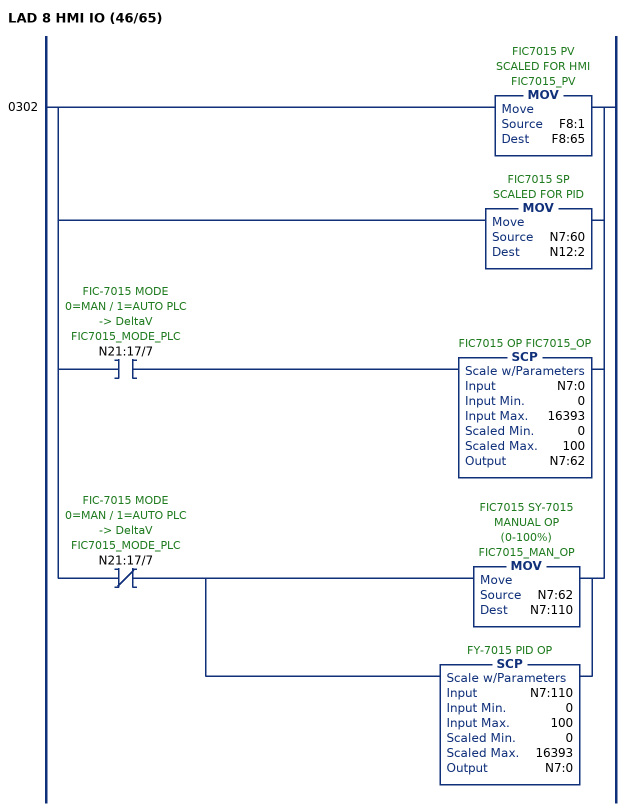
% Rung: 302 %
SOR BST MOV F8:1 F8:65 NXB MOV N7:60 N12:2 NXB XIC N21:17/7 SCP N7:0 0 16393 0 100 N7:62 NXB XIO N21:17/7 BST MOV N7:62 N7:110 NXB SCP N7:110 0 100 0 16393 N7:0 BND BND EOR
%   F8:1  FT_7010_SCI  "FT-7010 SCALED INPUT" %
%   F8:65  FIC7015_PV  "FIC7015 PV SCALED FOR HMI" %
%   N7:60  FIC7015_SP  "FIC7015 SP" %
%   N12:2  "FIC7015 SP SCALED FOR PID" %
%   N21:17/7  FIC7015_MODE_PLC  "FIC-7015 MODE 0=MAN / 1=AUTO PLC -> DeltaV" %
%   N7:0  "FY-7015 PID OP" %
%   N7:62  FIC7015_OP  "FIC7015 OP" %
%   N7:110  FIC7015_MAN_OP  "FIC7015 SY-7015 MANUAL OP (0-100%)" %

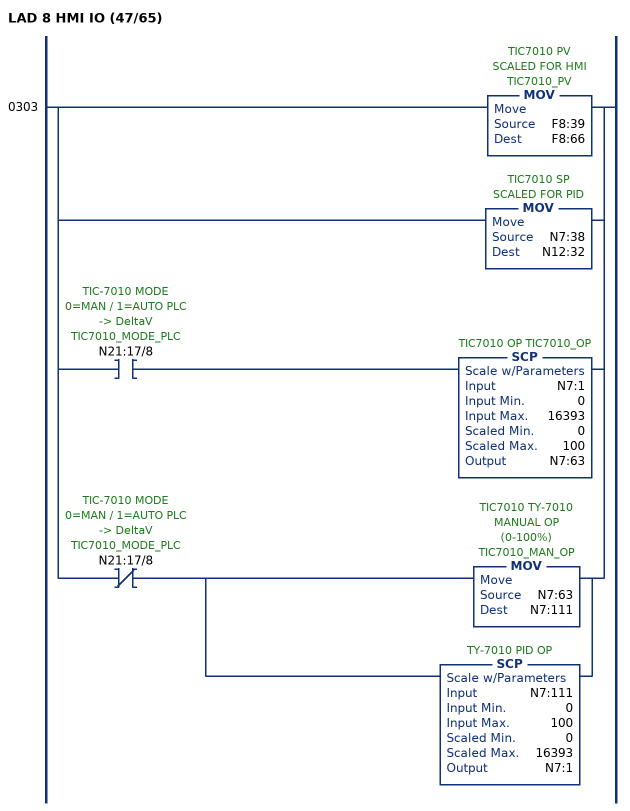
% Rung: 303 %
SOR BST MOV F8:39 F8:66 NXB MOV N7:38 N12:32 NXB XIC N21:17/8 SCP N7:1 0 16393 0 100 N7:63 NXB XIO N21:17/8 BST MOV N7:63 N7:111 NXB SCP N7:111 0 100 0 16393 N7:1 BND BND EOR
%   F8:39  TT_7010_SCI  "TT-7010 SCALED INPUT" %
%   F8:66  TIC7010_PV  "TIC7010 PV SCALED FOR HMI" %
%   N7:38  TIC7010_SP  "TIC7010 SP" %
%   N12:32  "TIC7010 SP SCALED FOR PID" %
%   N21:17/8  TIC7010_MODE_PLC  "TIC-7010 MODE 0=MAN / 1=AUTO PLC -> DeltaV" %
%   N7:1  "TY-7010 PID OP" %
%   N7:63  TIC7010_OP  "TIC7010 OP" %
%   N7:111  TIC7010_MAN_OP  "TIC7010 TY-7010 MANUAL OP (0-100%)" %

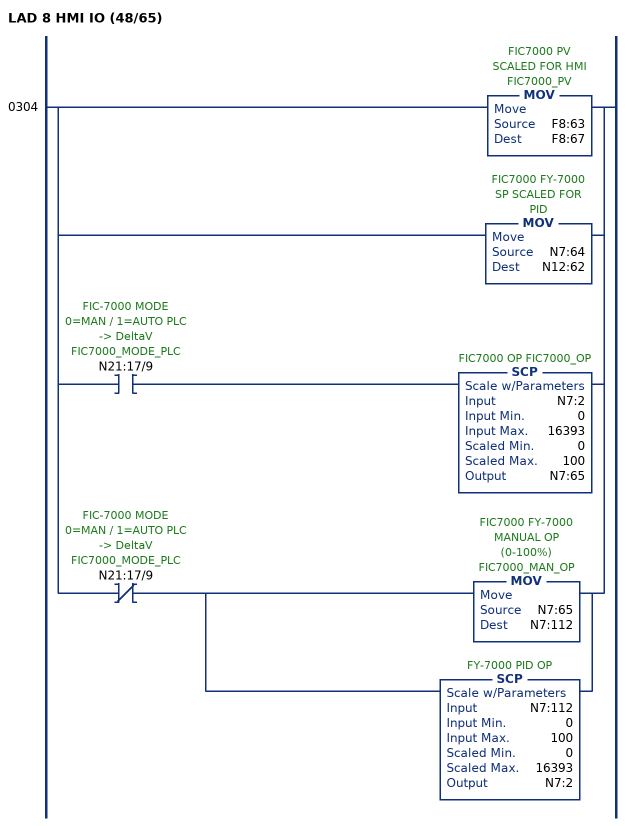
% Rung: 304 %
SOR BST MOV F8:63 F8:67 NXB MOV N7:64 N12:62 NXB XIC N21:17/9 SCP N7:2 0 16393 0 100 N7:65 NXB XIO N21:17/9 BST MOV N7:65 N7:112 NXB SCP N7:112 0 100 0 16393 N7:2 BND BND EOR
%   F8:63  PT_7026_SCI  "PT-7026 SCALED INPUT" %
%   F8:67  FIC7000_PV  "FIC7000 PV SCALED FOR HMI" %
%   N7:64  FIC7000_SP  "FIC7000 SP" %
%   N12:62  "FIC7000 FY-7000 SP SCALED FOR PID" %
%   N21:17/9  FIC7000_MODE_PLC  "FIC-7000 MODE 0=MAN / 1=AUTO PLC -> DeltaV" %
%   N7:2  "FY-7000 PID OP" %
%   N7:65  FIC7000_OP  "FIC7000 OP" %
%   N7:112  FIC7000_MAN_OP  "FIC7000 FY-7000 MANUAL OP (0-100%)" %

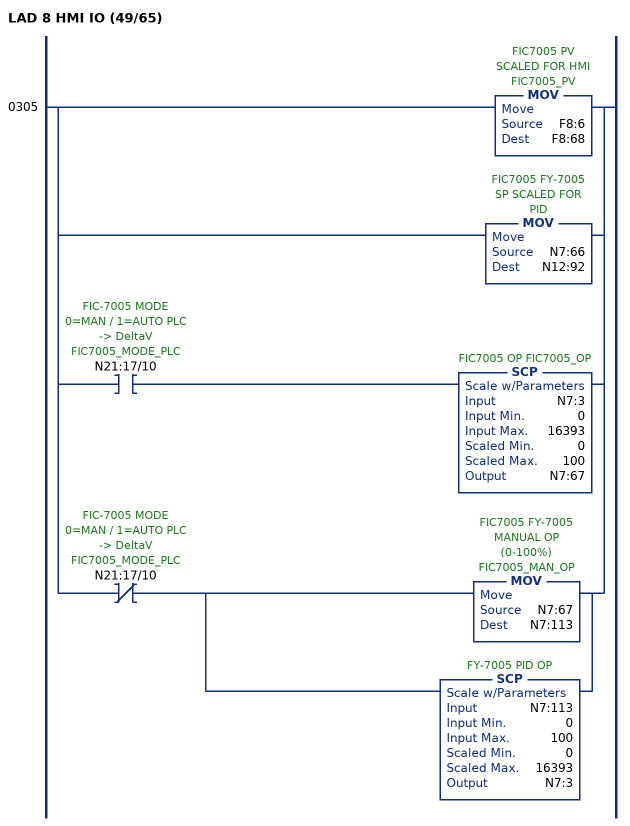
% Rung: 305 %
SOR BST MOV F8:6 F8:68 NXB MOV N7:66 N12:92 NXB XIC N21:17/10 SCP N7:3 0 16393 0 100 N7:67 NXB XIO N21:17/10 BST MOV N7:67 N7:113 NXB SCP N7:113 0 100 0 16393 N7:3 BND BND EOR
%   F8:6  FT_7005_SCI  "FT-7005 SCALED INPUT" %
%   F8:68  FIC7005_PV  "FIC7005 PV SCALED FOR HMI" %
%   N7:66  FIC7005_SP  "FIC7005 SP" %
%   N12:92  "FIC7005 FY-7005 SP SCALED FOR PID" %
%   N21:17/10  FIC7005_MODE_PLC  "FIC-7005 MODE 0=MAN / 1=AUTO PLC -> DeltaV" %
%   N7:3  "FY-7005 PID OP" %
%   N7:67  FIC7005_OP  "FIC7005 OP" %
%   N7:113  FIC7005_MAN_OP  "FIC7005 FY-7005 MANUAL OP (0-100%)" %

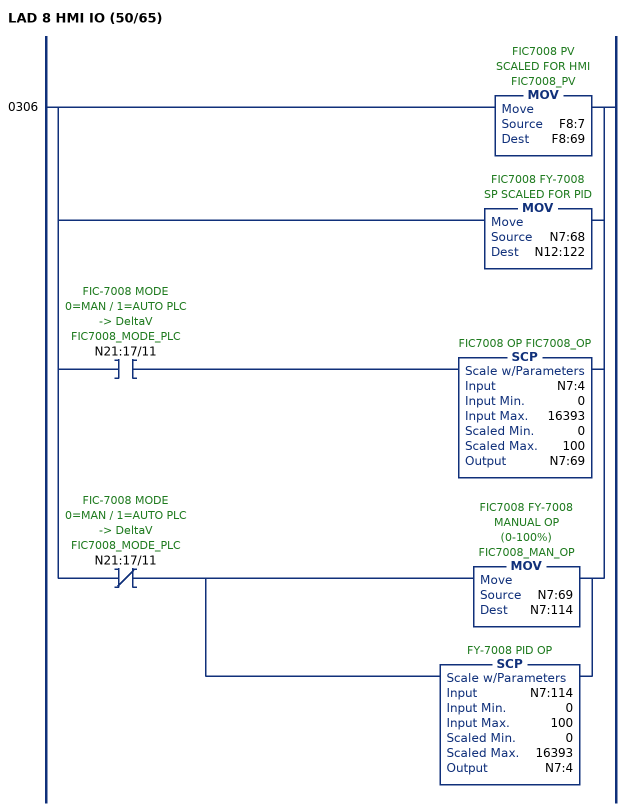
% Rung: 306 %
SOR BST MOV F8:7 F8:69 NXB MOV N7:68 N12:122 NXB XIC N21:17/11 SCP N7:4 0 16393 0 100 N7:69 NXB XIO N21:17/11 BST MOV N7:69 N7:114 NXB SCP N7:114 0 100 0 16393 N7:4 BND BND EOR
%   F8:7  FT_7008_SCI  "FT-7008 SCALED INPUT" %
%   F8:69  FIC7008_PV  "FIC7008 PV SCALED FOR HMI" %
%   N7:68  FIC7008_SP  "FIC7008 SP" %
%   N12:122  "FIC7008 FY-7008 SP SCALED FOR PID" %
%   N21:17/11  FIC7008_MODE_PLC  "FIC-7008 MODE 0=MAN / 1=AUTO PLC -> DeltaV" %
%   N7:4  "FY-7008 PID OP" %
%   N7:69  FIC7008_OP  "FIC7008 OP" %
%   N7:114  FIC7008_MAN_OP  "FIC7008 FY-7008 MANUAL OP (0-100%)" %

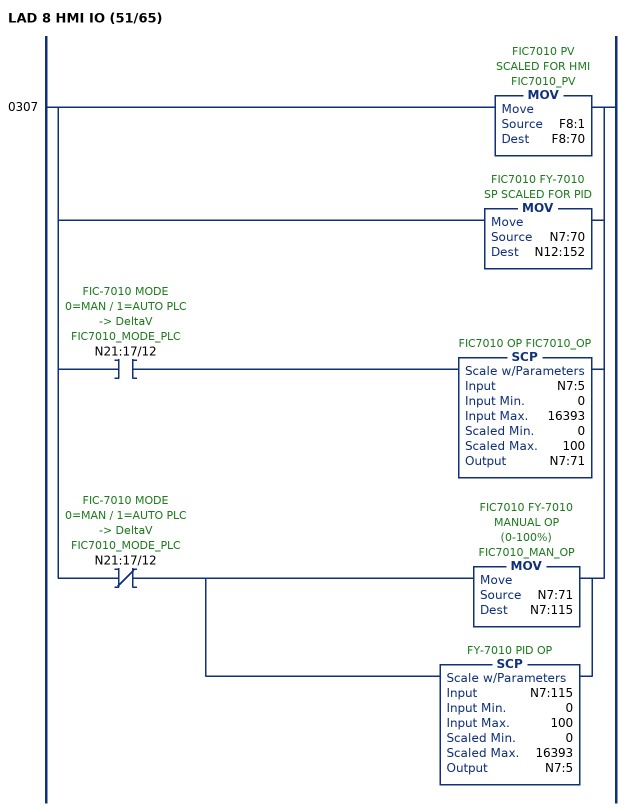
% Rung: 307 %
SOR BST MOV F8:1 F8:70 NXB MOV N7:70 N12:152 NXB XIC N21:17/12 SCP N7:5 0 16393 0 100 N7:71 NXB XIO N21:17/12 BST MOV N7:71 N7:115 NXB SCP N7:115 0 100 0 16393 N7:5 BND BND EOR
%   F8:1  FT_7010_SCI  "FT-7010 SCALED INPUT" %
%   F8:70  FIC7010_PV  "FIC7010 PV SCALED FOR HMI" %
%   N7:70  FIC7010_SP  "FIC7010 SP" %
%   N12:152  "FIC7010 FY-7010 SP SCALED FOR PID" %
%   N21:17/12  FIC7010_MODE_PLC  "FIC-7010 MODE 0=MAN / 1=AUTO PLC -> DeltaV" %
%   N7:5  "FY-7010 PID OP" %
%   N7:71  FIC7010_OP  "FIC7010 OP" %
%   N7:115  FIC7010_MAN_OP  "FIC7010 FY-7010 MANUAL OP (0-100%)" %

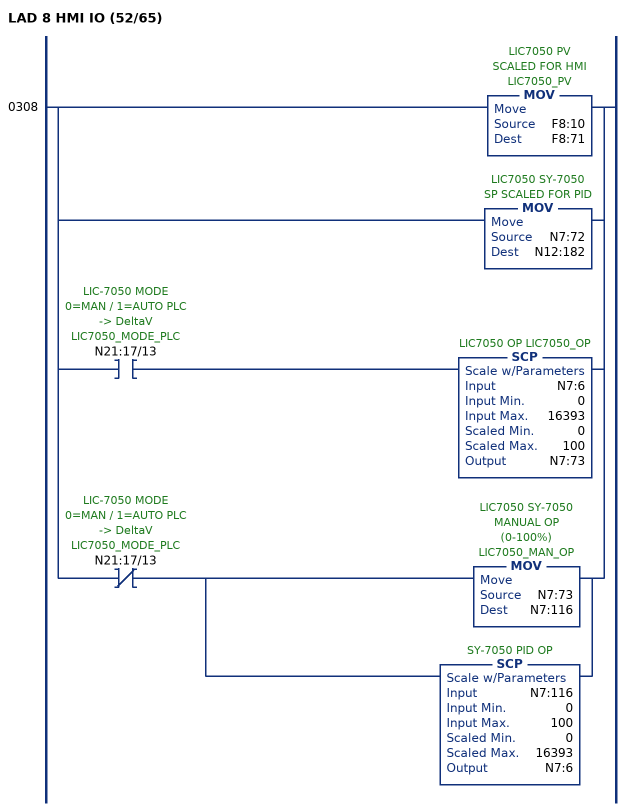
% Rung: 308 %
SOR BST MOV F8:10 F8:71 NXB MOV N7:72 N12:182 NXB XIC N21:17/13 SCP N7:6 0 16393 0 100 N7:73 NXB XIO N21:17/13 BST MOV N7:73 N7:116 NXB SCP N7:116 0 100 0 16393 N7:6 BND BND EOR
%   F8:10  LT_7050_SCI  "LT-7050 SCALED INPUT" %
%   F8:71  LIC7050_PV  "LIC7050 PV SCALED FOR HMI" %
%   N7:72  LIC7050_SP  "LIC7050 SP" %
%   N12:182  "LIC7050 SY-7050 SP SCALED FOR PID" %
%   N21:17/13  LIC7050_MODE_PLC  "LIC-7050 MODE 0=MAN / 1=AUTO PLC -> DeltaV" %
%   N7:6  "SY-7050 PID OP" %
%   N7:73  LIC7050_OP  "LIC7050 OP" %
%   N7:116  LIC7050_MAN_OP  "LIC7050 SY-7050 MANUAL OP (0-100%)" %

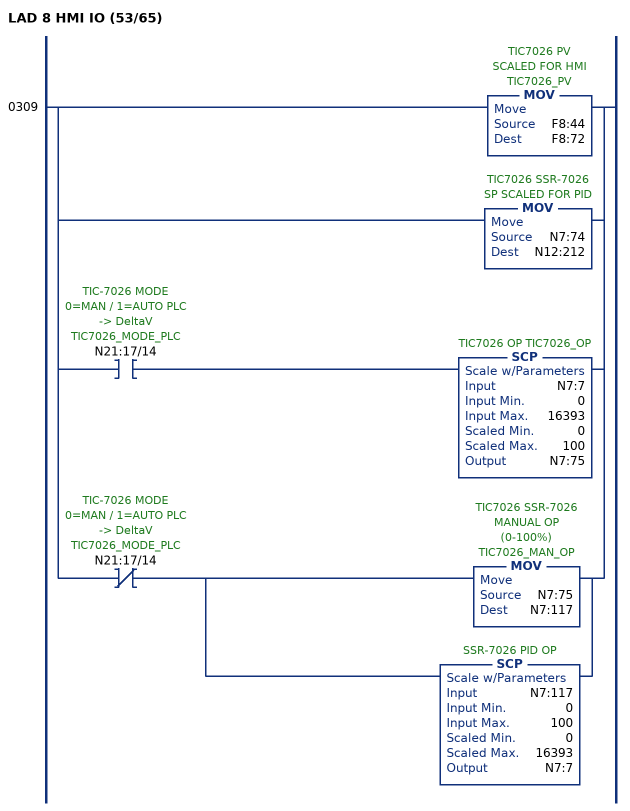
% Rung: 309 %
SOR BST MOV F8:44 F8:72 NXB MOV N7:74 N12:212 NXB XIC N21:17/14 SCP N7:7 0 16393 0 100 N7:75 NXB XIO N21:17/14 BST MOV N7:75 N7:117 NXB SCP N7:117 0 100 0 16393 N7:7 BND BND EOR
%   F8:44  TT_7026_SCI  "TT-7026 SCALED INPUT" %
%   F8:72  TIC7026_PV  "TIC7026 PV SCALED FOR HMI" %
%   N7:74  TIC7026_SP  "TIC7026 SP" %
%   N12:212  "TIC7026 SSR-7026 SP SCALED FOR PID" %
%   N21:17/14  TIC7026_MODE_PLC  "TIC-7026 MODE 0=MAN / 1=AUTO PLC -> DeltaV" %
%   N7:7  "SSR-7026 PID OP" %
%   N7:75  TIC7026_OP  "TIC7026 OP" %
%   N7:117  TIC7026_MAN_OP  "TIC7026 SSR-7026 MANUAL OP (0-100%)" %

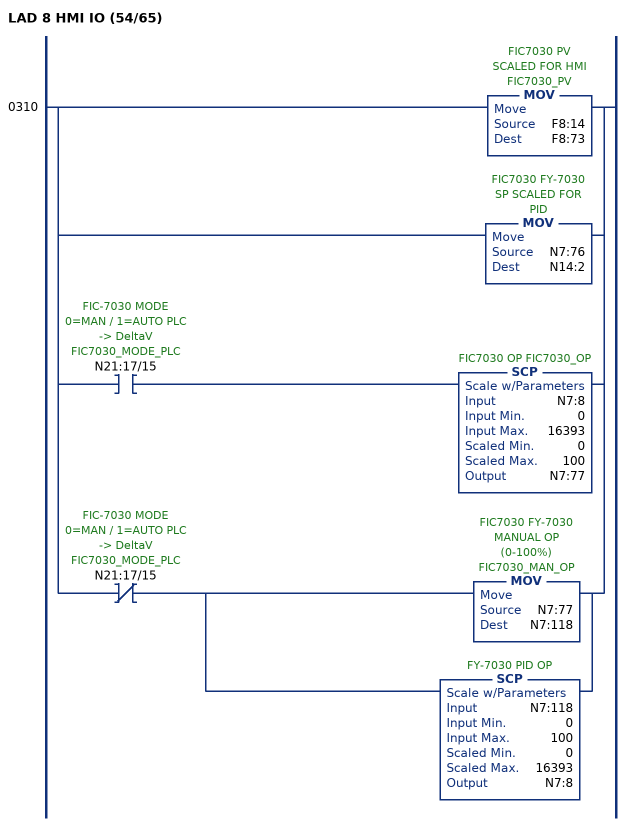
% Rung: 310 %
SOR BST MOV F8:14 F8:73 NXB MOV N7:76 N14:2 NXB XIC N21:17/15 SCP N7:8 0 16393 0 100 N7:77 NXB XIO N21:17/15 BST MOV N7:77 N7:118 NXB SCP N7:118 0 100 0 16393 N7:8 BND BND EOR
%   F8:14  FT_7030_SCI  "FT-7030 SCALED INPUT" %
%   F8:73  FIC7030_PV  "FIC7030 PV SCALED FOR HMI" %
%   N7:76  FIC7030_SP  "FIC7030 SP" %
%   N14:2  "FIC7030 FY-7030 SP SCALED FOR PID" %
%   N21:17/15  FIC7030_MODE_PLC  "FIC-7030 MODE 0=MAN / 1=AUTO PLC -> DeltaV" %
%   N7:8  "FY-7030 PID OP" %
%   N7:77  FIC7030_OP  "FIC7030 OP" %
%   N7:118  FIC7030_MAN_OP  "FIC7030 FY-7030 MANUAL OP (0-100%)" %

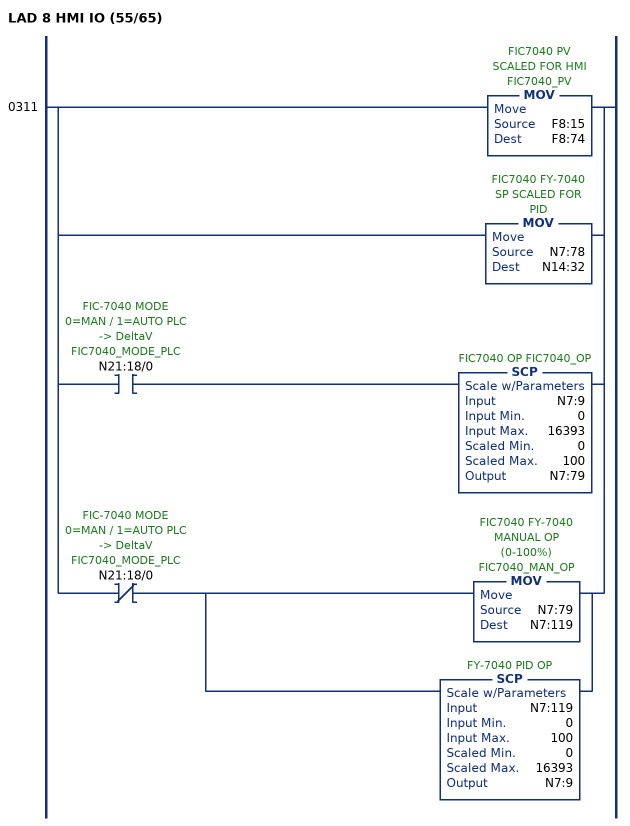
% Rung: 311 %
SOR BST MOV F8:15 F8:74 NXB MOV N7:78 N14:32 NXB XIC N21:18/0 SCP N7:9 0 16393 0 100 N7:79 NXB XIO N21:18/0 BST MOV N7:79 N7:119 NXB SCP N7:119 0 100 0 16393 N7:9 BND BND EOR
%   F8:15  FT_7040_SCI  "FT-7040 SCALED INPUT" %
%   F8:74  FIC7040_PV  "FIC7040 PV SCALED FOR HMI" %
%   N7:78  FIC7040_SP  "FIC7040 SP" %
%   N14:32  "FIC7040 FY-7040 SP SCALED FOR PID" %
%   N21:18/0  FIC7040_MODE_PLC  "FIC-7040 MODE 0=MAN / 1=AUTO PLC -> DeltaV" %
%   N7:9  "FY-7040 PID OP" %
%   N7:79  FIC7040_OP  "FIC7040 OP" %
%   N7:119  FIC7040_MAN_OP  "FIC7040 FY-7040 MANUAL OP (0-100%)" %

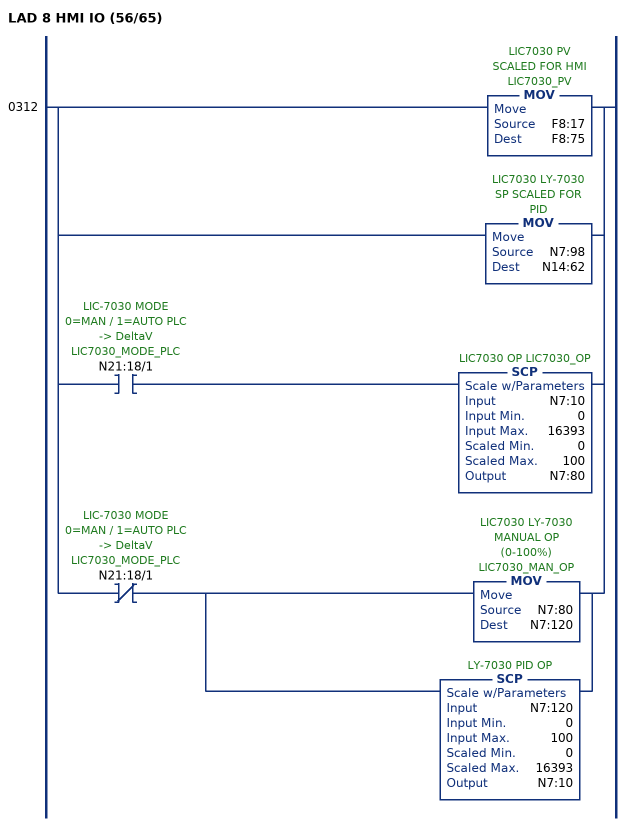
% Rung: 312 %
SOR BST MOV F8:17 F8:75 NXB MOV N7:98 N14:62 NXB XIC N21:18/1 SCP N7:10 0 16393 0 100 N7:80 NXB XIO N21:18/1 BST MOV N7:80 N7:120 NXB SCP N7:120 0 100 0 16393 N7:10 BND BND EOR
%   F8:17  LT_7030_SCI  "LT-7030 SCALED INPUT" %
%   F8:75  LIC7030_PV  "LIC7030 PV SCALED FOR HMI" %
%   N7:98  LIC7030_SP  "LIC7030 SP" %
%   N14:62  "LIC7030 LY-7030 SP SCALED FOR PID" %
%   N21:18/1  LIC7030_MODE_PLC  "LIC-7030 MODE 0=MAN / 1=AUTO PLC -> DeltaV" %
%   N7:10  "LY-7030 PID OP" %
%   N7:80  LIC7030_OP  "LIC7030 OP" %
%   N7:120  LIC7030_MAN_OP  "LIC7030 LY-7030 MANUAL OP (0-100%)" %

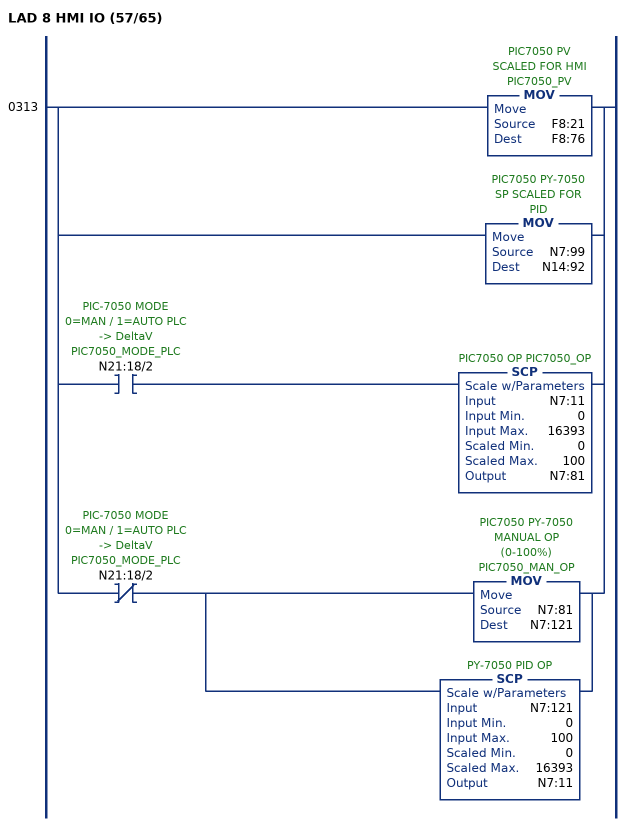
% Rung: 313 %
SOR BST MOV F8:21 F8:76 NXB MOV N7:99 N14:92 NXB XIC N21:18/2 SCP N7:11 0 16393 0 100 N7:81 NXB XIO N21:18/2 BST MOV N7:81 N7:121 NXB SCP N7:121 0 100 0 16393 N7:11 BND BND EOR
%   F8:21  PT_7050_SCI  "PT-7050 SCALED INPUT" %
%   F8:76  PIC7050_PV  "PIC7050 PV SCALED FOR HMI" %
%   N7:99  PIC7050_SP  "PIC7050 SP" %
%   N14:92  "PIC7050 PY-7050 SP SCALED FOR PID" %
%   N21:18/2  PIC7050_MODE_PLC  "PIC-7050 MODE 0=MAN / 1=AUTO PLC -> DeltaV" %
%   N7:11  "PY-7050 PID OP" %
%   N7:81  PIC7050_OP  "PIC7050 OP" %
%   N7:121  PIC7050_MAN_OP  "PIC7050 PY-7050 MANUAL OP (0-100%)" %

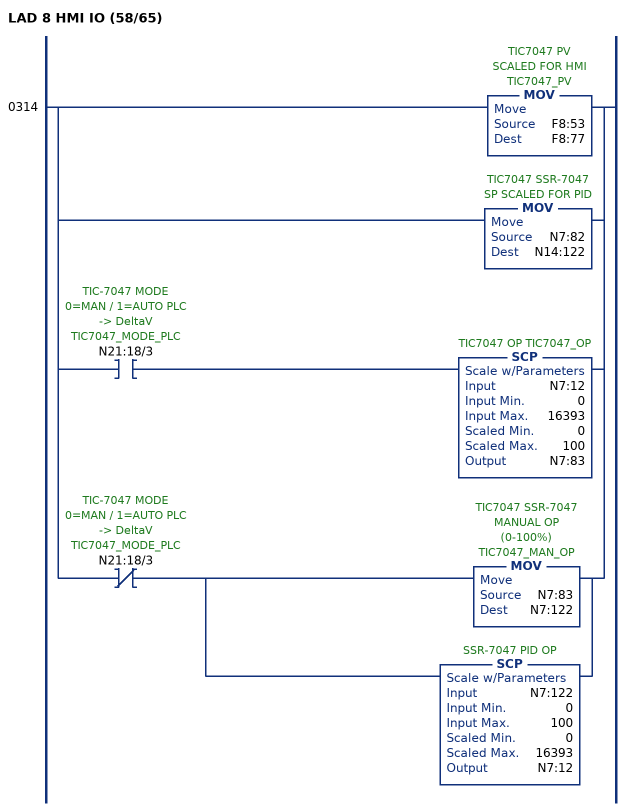
% Rung: 314 %
SOR BST MOV F8:53 F8:77 NXB MOV N7:82 N14:122 NXB XIC N21:18/3 SCP N7:12 0 16393 0 100 N7:83 NXB XIO N21:18/3 BST MOV N7:83 N7:122 NXB SCP N7:122 0 100 0 16393 N7:12 BND BND EOR
%   F8:53  TT_7047_SCI  "TT-7047 SCALED INPUT" %
%   F8:77  TIC7047_PV  "TIC7047 PV SCALED FOR HMI" %
%   N7:82  TIC7047_SP  "TIC7047 SP" %
%   N14:122  "TIC7047 SSR-7047 SP SCALED FOR PID" %
%   N21:18/3  TIC7047_MODE_PLC  "TIC-7047 MODE 0=MAN / 1=AUTO PLC -> DeltaV" %
%   N7:12  "SSR-7047 PID OP" %
%   N7:83  TIC7047_OP  "TIC7047 OP" %
%   N7:122  TIC7047_MAN_OP  "TIC7047 SSR-7047 MANUAL OP (0-100%)" %

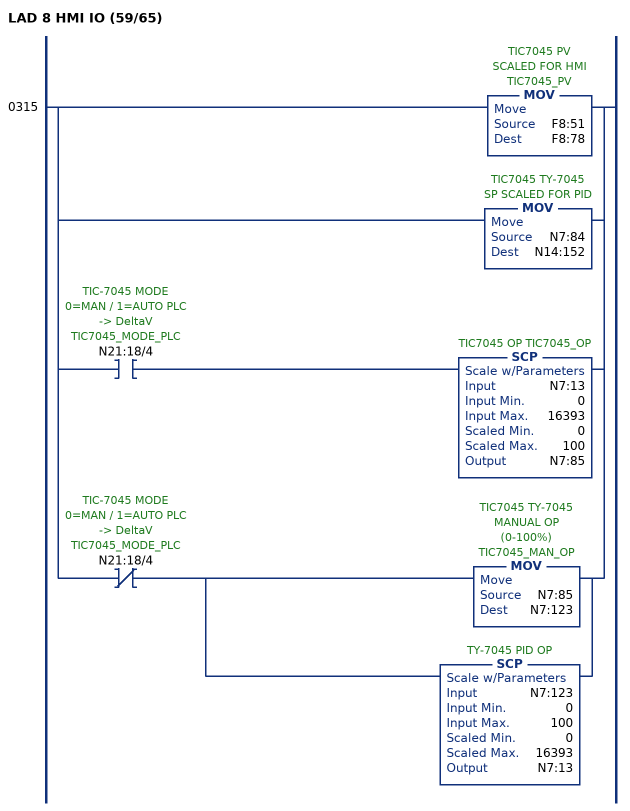
% Rung: 315 %
SOR BST MOV F8:51 F8:78 NXB MOV N7:84 N14:152 NXB XIC N21:18/4 SCP N7:13 0 16393 0 100 N7:85 NXB XIO N21:18/4 BST MOV N7:85 N7:123 NXB SCP N7:123 0 100 0 16393 N7:13 BND BND EOR
%   F8:51  TT_7045_SCI  "TT-7045 SCALED INPUT" %
%   F8:78  TIC7045_PV  "TIC7045 PV SCALED FOR HMI" %
%   N7:84  TIC7045_SP  "TIC7045 SP" %
%   N14:152  "TIC7045 TY-7045 SP SCALED FOR PID" %
%   N21:18/4  TIC7045_MODE_PLC  "TIC-7045 MODE 0=MAN / 1=AUTO PLC -> DeltaV" %
%   N7:13  "TY-7045 PID OP" %
%   N7:85  TIC7045_OP  "TIC7045 OP" %
%   N7:123  TIC7045_MAN_OP  "TIC7045 TY-7045 MANUAL OP (0-100%)" %

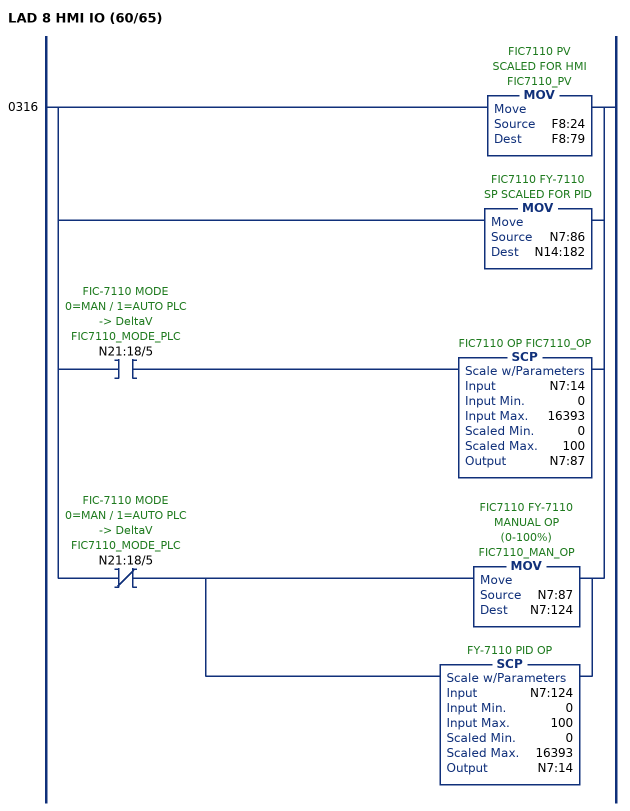
% Rung: 316 %
SOR BST MOV F8:24 F8:79 NXB MOV N7:86 N14:182 NXB XIC N21:18/5 SCP N7:14 0 16393 0 100 N7:87 NXB XIO N21:18/5 BST MOV N7:87 N7:124 NXB SCP N7:124 0 100 0 16393 N7:14 BND BND EOR
%   F8:24  FT_7110_SCI  "FT-7110 SCALED INPUT" %
%   F8:79  FIC7110_PV  "FIC7110 PV SCALED FOR HMI" %
%   N7:86  FIC7110_SP  "FIC7110 SP" %
%   N14:182  "FIC7110 FY-7110 SP SCALED FOR PID" %
%   N21:18/5  FIC7110_MODE_PLC  "FIC-7110 MODE 0=MAN / 1=AUTO PLC -> DeltaV" %
%   N7:14  "FY-7110 PID OP" %
%   N7:87  FIC7110_OP  "FIC7110 OP" %
%   N7:124  FIC7110_MAN_OP  "FIC7110 FY-7110 MANUAL OP (0-100%)" %

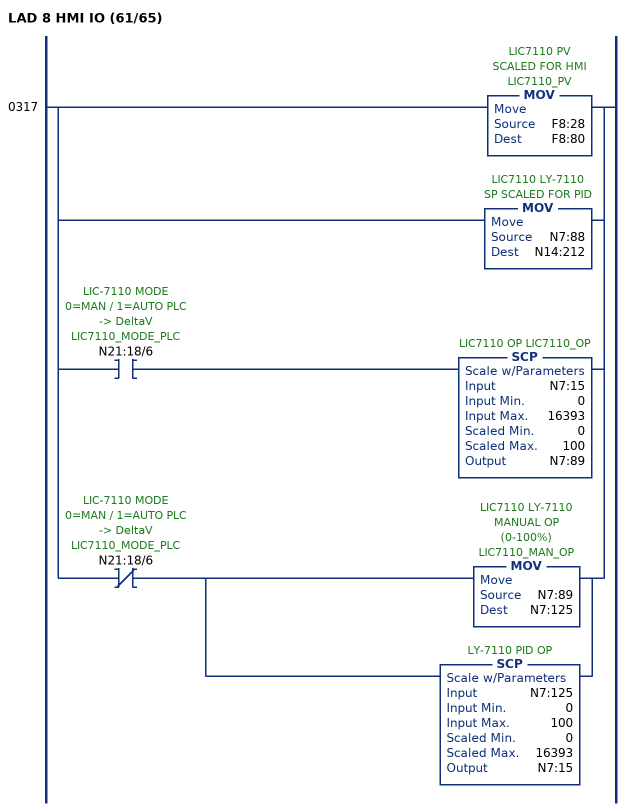
% Rung: 317 %
SOR BST MOV F8:28 F8:80 NXB MOV N7:88 N14:212 NXB XIC N21:18/6 SCP N7:15 0 16393 0 100 N7:89 NXB XIO N21:18/6 BST MOV N7:89 N7:125 NXB SCP N7:125 0 100 0 16393 N7:15 BND BND EOR
%   F8:28  LT_7110_SCI  "LT-7110 SCALED INPUT" %
%   F8:80  LIC7110_PV  "LIC7110 PV SCALED FOR HMI" %
%   N7:88  LIC7110_SP  "LIC7110 SP" %
%   N14:212  "LIC7110 LY-7110 SP SCALED FOR PID" %
%   N21:18/6  LIC7110_MODE_PLC  "LIC-7110 MODE 0=MAN / 1=AUTO PLC -> DeltaV" %
%   N7:15  "LY-7110 PID OP" %
%   N7:89  LIC7110_OP  "LIC7110 OP" %
%   N7:125  LIC7110_MAN_OP  "LIC7110 LY-7110 MANUAL OP (0-100%)" %

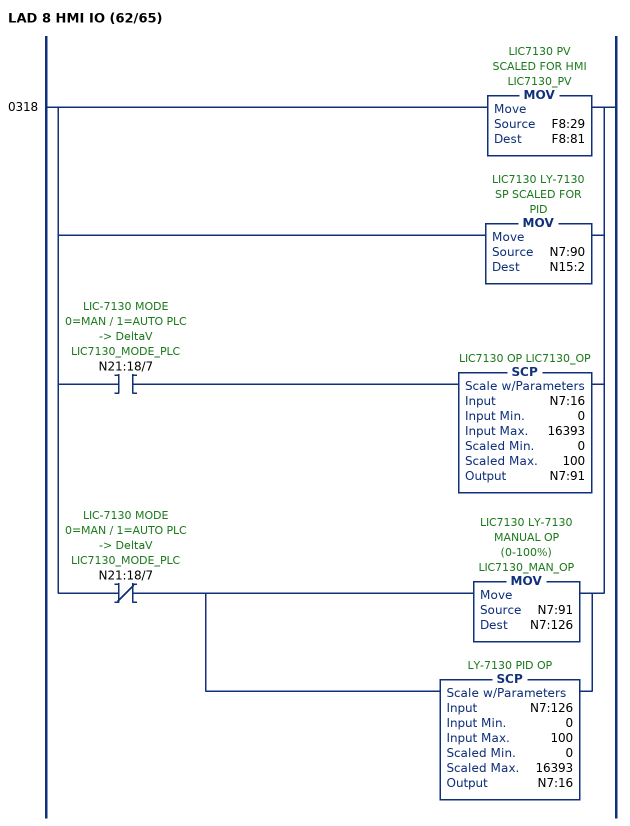
% Rung: 318 %
SOR BST MOV F8:29 F8:81 NXB MOV N7:90 N15:2 NXB XIC N21:18/7 SCP N7:16 0 16393 0 100 N7:91 NXB XIO N21:18/7 BST MOV N7:91 N7:126 NXB SCP N7:126 0 100 0 16393 N7:16 BND BND EOR
%   F8:29  LT_7130_SCI  "LT-7130 SCALED INPUT" %
%   F8:81  LIC7130_PV  "LIC7130 PV SCALED FOR HMI" %
%   N7:90  LIC7130_SP  "LIC7130 SP" %
%   N15:2  "LIC7130 LY-7130 SP SCALED FOR PID" %
%   N21:18/7  LIC7130_MODE_PLC  "LIC-7130 MODE 0=MAN / 1=AUTO PLC -> DeltaV" %
%   N7:16  "LY-7130 PID OP" %
%   N7:91  LIC7130_OP  "LIC7130 OP" %
%   N7:126  LIC7130_MAN_OP  "LIC7130 LY-7130 MANUAL OP (0-100%)" %

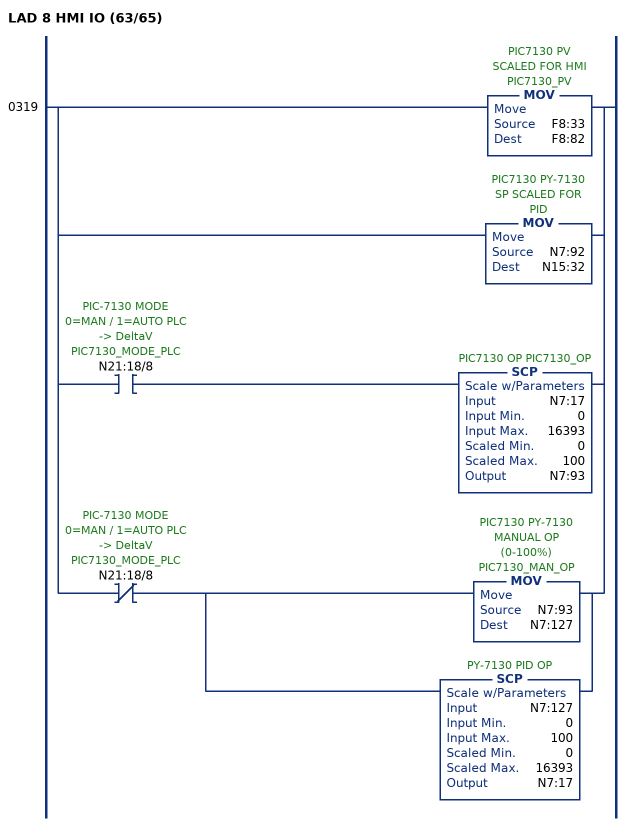
% Rung: 319 %
SOR BST MOV F8:33 F8:82 NXB MOV N7:92 N15:32 NXB XIC N21:18/8 SCP N7:17 0 16393 0 100 N7:93 NXB XIO N21:18/8 BST MOV N7:93 N7:127 NXB SCP N7:127 0 100 0 16393 N7:17 BND BND EOR
%   F8:33  PT_7130_SCI  "PT-7130 SCALED INPUT" %
%   F8:82  PIC7130_PV  "PIC7130 PV SCALED FOR HMI" %
%   N7:92  PIC7130_SP  "PIC7130 SP" %
%   N15:32  "PIC7130 PY-7130 SP SCALED FOR PID" %
%   N21:18/8  PIC7130_MODE_PLC  "PIC-7130 MODE 0=MAN / 1=AUTO PLC -> DeltaV" %
%   N7:17  "PY-7130 PID OP" %
%   N7:93  PIC7130_OP  "PIC7130 OP" %
%   N7:127  PIC7130_MAN_OP  "PIC7130 PY-7130 MANUAL OP (0-100%)" %

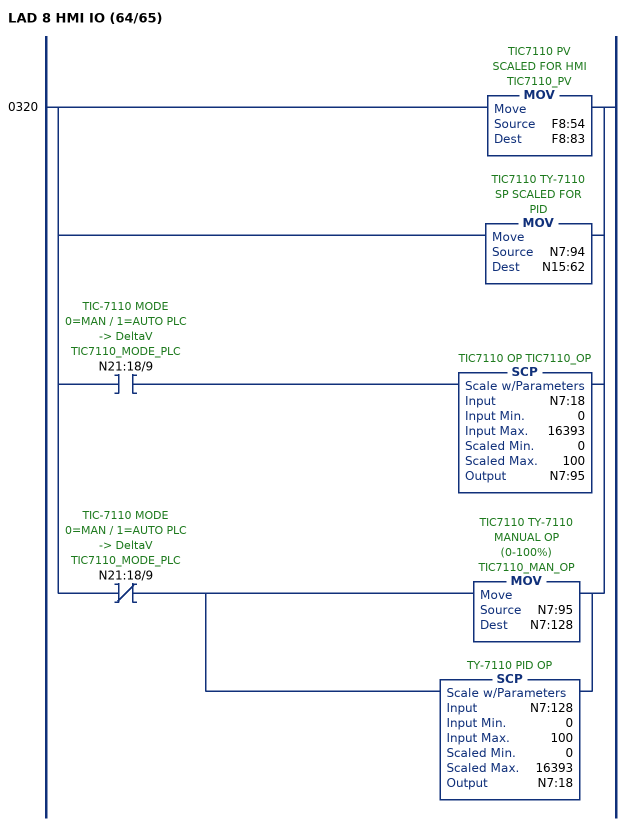
% Rung: 320 %
SOR BST MOV F8:54 F8:83 NXB MOV N7:94 N15:62 NXB XIC N21:18/9 SCP N7:18 0 16393 0 100 N7:95 NXB XIO N21:18/9 BST MOV N7:95 N7:128 NXB SCP N7:128 0 100 0 16393 N7:18 BND BND EOR
%   F8:54  TT_7110_SCI  "TT-7110 SCALED INPUT" %
%   F8:83  TIC7110_PV  "TIC7110 PV SCALED FOR HMI" %
%   N7:94  TIC7110_SP  "TIC7110 SP" %
%   N15:62  "TIC7110 TY-7110 SP SCALED FOR PID" %
%   N21:18/9  TIC7110_MODE_PLC  "TIC-7110 MODE 0=MAN / 1=AUTO PLC -> DeltaV" %
%   N7:18  "TY-7110 PID OP" %
%   N7:95  TIC7110_OP  "TIC7110 OP" %
%   N7:128  TIC7110_MAN_OP  "TIC7110 TY-7110 MANUAL OP (0-100%)" %

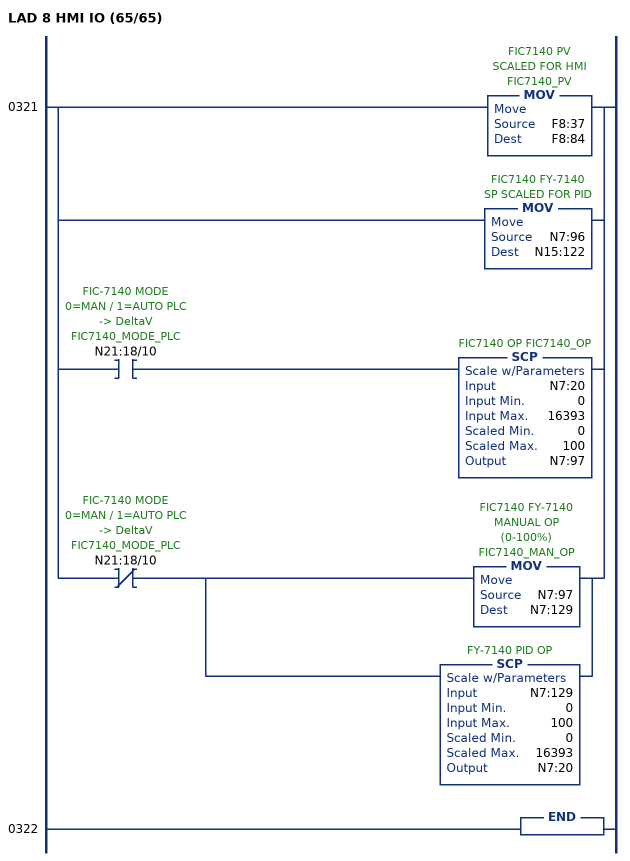
% Rung: 321 %
SOR BST MOV F8:37 F8:84 NXB MOV N7:96 N15:122 NXB XIC N21:18/10 SCP N7:20 0 16393 0 100 N7:97 NXB XIO N21:18/10 BST MOV N7:97 N7:129 NXB SCP N7:129 0 100 0 16393 N7:20 BND BND EOR
%   F8:37  FT_7140_SCI  "FT-7140 SCALED INPUT" %
%   F8:84  FIC7140_PV  "FIC7140 PV SCALED FOR HMI" %
%   N7:96  FIC7140_SP  "FIC7140 SP" %
%   N15:122  "FIC7140 FY-7140 SP SCALED FOR PID" %
%   N21:18/10  FIC7140_MODE_PLC  "FIC-7140 MODE 0=MAN / 1=AUTO PLC -> DeltaV" %
%   N7:20  "FY-7140 PID OP" %
%   N7:97  FIC7140_OP  "FIC7140 OP" %
%   N7:129  FIC7140_MAN_OP  "FIC7140 FY-7140 MANUAL OP (0-100%)" %
% Rung: 322 %
SOR END EOR

LADDER 9 "LOOPS"
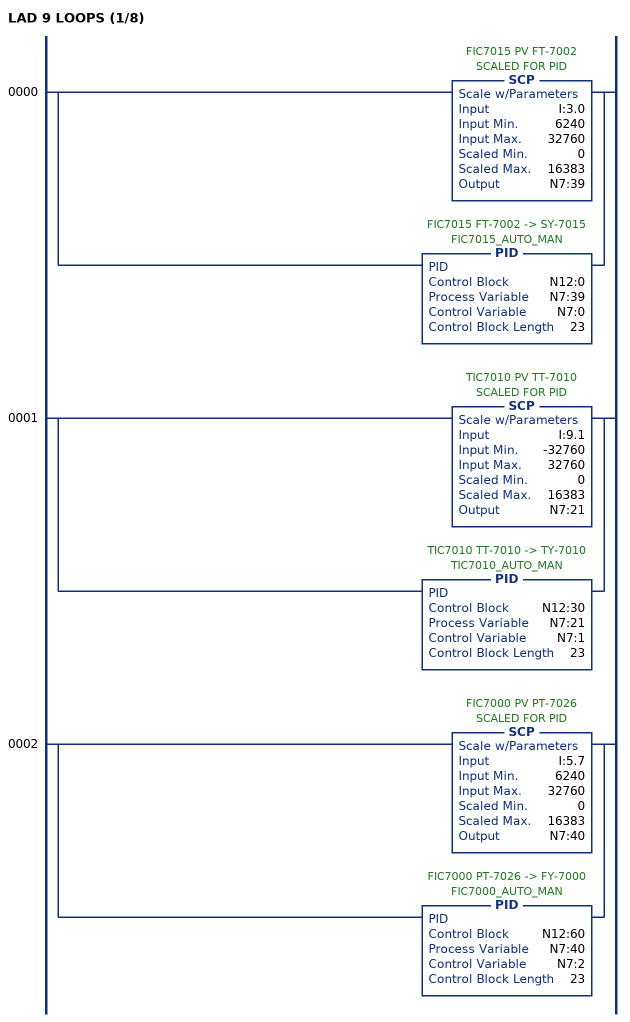
% Rung: 0 %
SOR BST SCP I:3.0 6240 32760 0 16383 N7:39 NXB PID N12:0 N7:39 N7:0 23 BND EOR
%   I:3.0  FT_7002  "FT-7002 ANALOG IN" %
%   N7:39  "FIC7015 PV FT-7002 SCALED FOR PID" %
%   N12:0  FIC7015_AUTO_MAN  "FIC7015 FT-7002 -> SY-7015" %
%   N7:0  "FY-7015 PID OP" %
% Rung: 1 %
SOR BST SCP I:9.1 -32760 32760 0 16383 N7:21 NXB PID N12:30 N7:21 N7:1 23 BND EOR
%   I:9.1  TT_7010  "TT-7010 ANALOG IN" %
%   N7:21  "TIC7010 PV TT-7010 SCALED FOR PID" %
%   N12:30  TIC7010_AUTO_MAN  "TIC7010 TT-7010 -> TY-7010" %
%   N7:1  "TY-7010 PID OP" %
% Rung: 2 %
SOR BST SCP I:5.7 6240 32760 0 16383 N7:40 NXB PID N12:60 N7:40 N7:2 23 BND EOR
%   I:5.7  PT_7026  "PT-7026 ANALOG IN" %
%   N7:40  "FIC7000 PV PT-7026 SCALED FOR PID" %
%   N12:60  FIC7000_AUTO_MAN  "FIC7000 PT-7026 -> FY-7000" %
%   N7:2  "FY-7000 PID OP" %

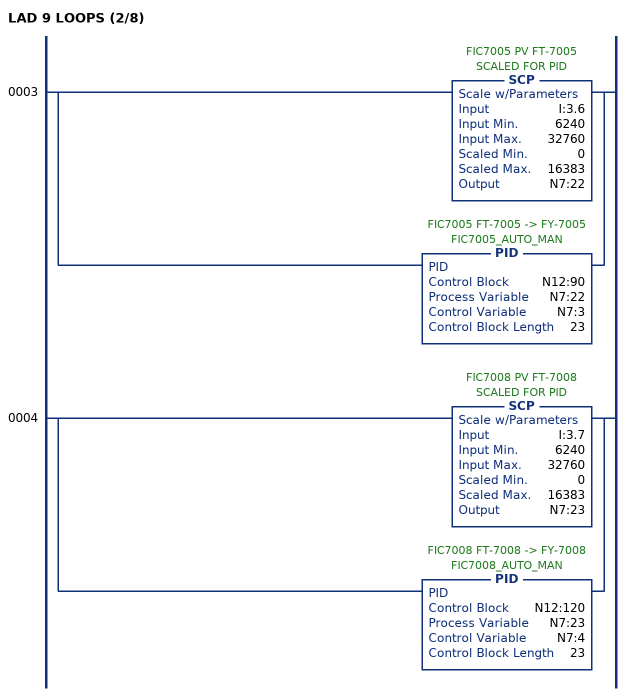
% Rung: 3 %
SOR BST SCP I:3.6 6240 32760 0 16383 N7:22 NXB PID N12:90 N7:22 N7:3 23 BND EOR
%   I:3.6  FT_7005  "FT-7005 ANALOG IN" %
%   N7:22  "FIC7005 PV FT-7005 SCALED FOR PID" %
%   N12:90  FIC7005_AUTO_MAN  "FIC7005 FT-7005 -> FY-7005" %
%   N7:3  "FY-7005 PID OP" %
% Rung: 4 %
SOR BST SCP I:3.7 6240 32760 0 16383 N7:23 NXB PID N12:120 N7:23 N7:4 23 BND EOR
%   I:3.7  FT_7008  "FT-7008 ANALOG IN" %
%   N7:23  "FIC7008 PV FT-7008 SCALED FOR PID" %
%   N12:120  FIC7008_AUTO_MAN  "FIC7008 FT-7008 -> FY-7008" %
%   N7:4  "FY-7008 PID OP" %

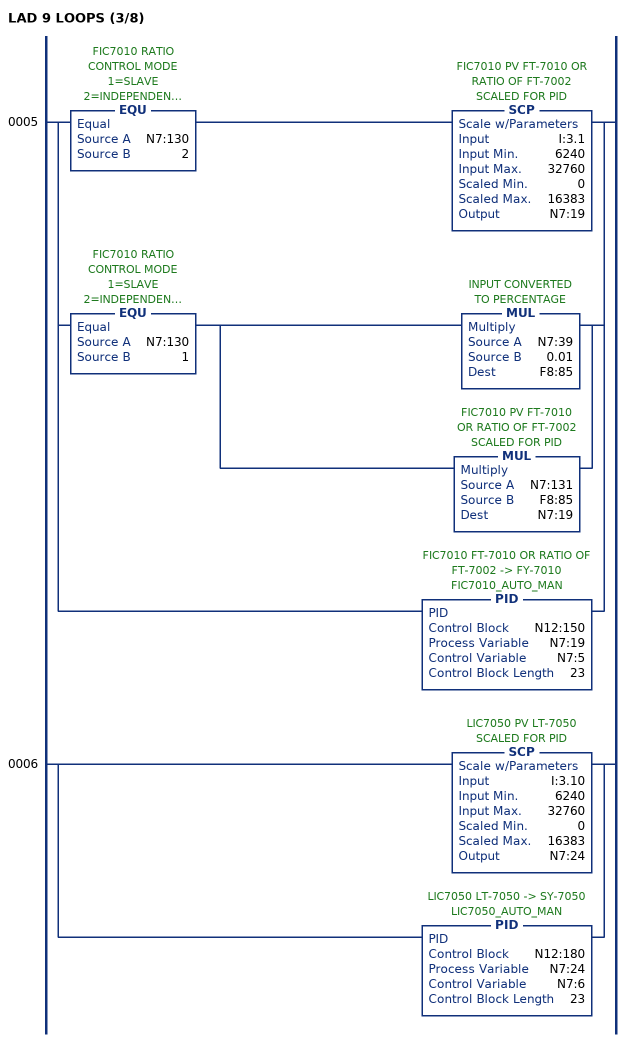
% Rung: 5 %
SOR BST EQU N7:130 2 SCP I:3.1 6240 32760 0 16383 N7:19 NXB EQU N7:130 1 BST MUL N7:39 0.01 F8:85 NXB MUL N7:131 F8:85 N7:19 BND NXB PID N12:150 N7:19 N7:5 23 BND EOR
%   N7:130  FIC7010_RATIO_MODE  "FIC7010 RATIO CONTROL MODE 1=SLAVE 2=INDEPENDENT" %
%   I:3.1  FT_7010  "FT-7010 ANALOG IN" %
%   N7:19  "FIC7010 PV FT-7010 OR RATIO OF FT-7002 SCALED FOR PID" %
%   N7:39  "FIC7015 PV FT-7002 SCALED FOR PID" %
%   F8:85  "INPUT CONVERTED TO PERCENTAGE" %
%   N7:131  FIC7010_RATIO_SP  "FIC7010 RATIO SP (0-100% OF FT-7002 FLOW)" %
%   N12:150  FIC7010_AUTO_MAN  "FIC7010 FT-7010 OR RATIO OF FT-7002 -> FY-7010" %
%   N7:5  "FY-7010 PID OP" %
% Rung: 6 %
SOR BST SCP I:3.10 6240 32760 0 16383 N7:24 NXB PID N12:180 N7:24 N7:6 23 BND EOR
%   I:3.10  LT_7050  "LT-7050 ANALOG IN" %
%   N7:24  "LIC7050 PV LT-7050 SCALED FOR PID" %
%   N12:180  LIC7050_AUTO_MAN  "LIC7050 LT-7050 -> SY-7050" %
%   N7:6  "SY-7050 PID OP" %

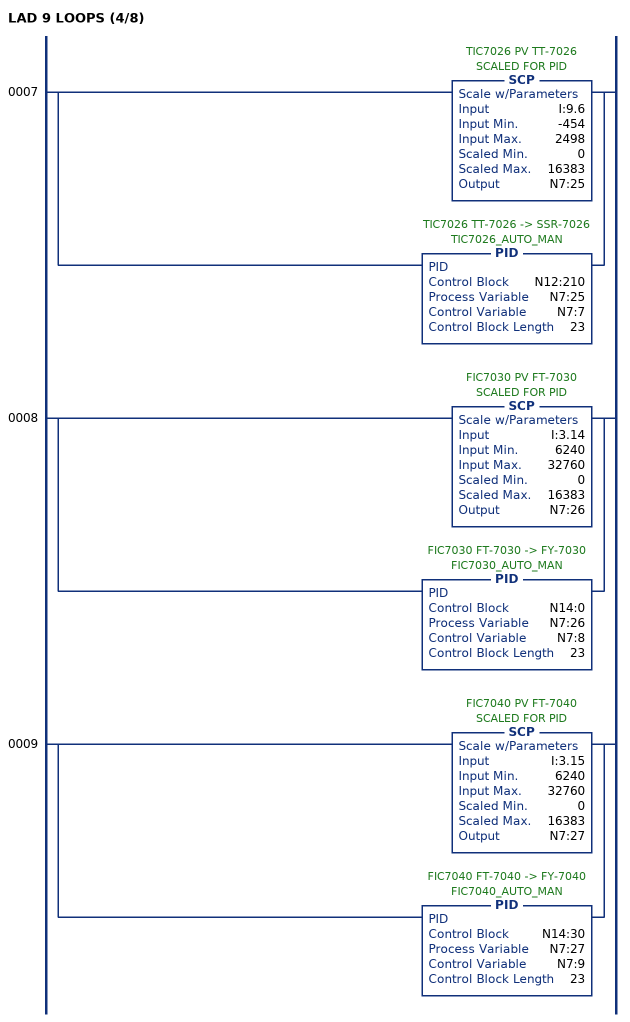
% Rung: 7 %
SOR BST SCP I:9.6 -454 2498 0 16383 N7:25 NXB PID N12:210 N7:25 N7:7 23 BND EOR
%   I:9.6  TT_7026  "TT-7026 ANALOG IN" %
%   N7:25  "TIC7026 PV TT-7026 SCALED FOR PID" %
%   N12:210  TIC7026_AUTO_MAN  "TIC7026 TT-7026 -> SSR-7026" %
%   N7:7  "SSR-7026 PID OP" %
% Rung: 8 %
SOR BST SCP I:3.14 6240 32760 0 16383 N7:26 NXB PID N14:0 N7:26 N7:8 23 BND EOR
%   I:3.14  FT_7030  "FT-7030 ANALOG IN" %
%   N7:26  "FIC7030 PV FT-7030 SCALED FOR PID" %
%   N14:0  FIC7030_AUTO_MAN  "FIC7030 FT-7030 -> FY-7030" %
%   N7:8  "FY-7030 PID OP" %
% Rung: 9 %
SOR BST SCP I:3.15 6240 32760 0 16383 N7:27 NXB PID N14:30 N7:27 N7:9 23 BND EOR
%   I:3.15  FT_7040  "FT-7040 ANALOG IN" %
%   N7:27  "FIC7040 PV FT-7040 SCALED FOR PID" %
%   N14:30  FIC7040_AUTO_MAN  "FIC7040 FT-7040 -> FY-7040" %
%   N7:9  "FY-7040 PID OP" %

